FUNCTION F_ConvertColorSpaceST
VAR_INPUT
END_VAR
VAR
END_VAR

END_FUNCTION

(* stored: Version 1.1.0.1, ProductVersion 3.1.4024.12
   POU F_ConvertColorSpaceST: Id {8afd784b-63f5-4640-a6cd-39ebc87076aa}, SpecialFunc None *)
